TYPE ST_PNOutput_GenControl :
STRUCT
	w_Status					:	WORD;
	w_Warnings					:	WORD;
	w_Faults					:	WORD;
	ui_GeneratorStatus			:	UINT;	
END_STRUCT
END_TYPE

(* stored: Version 1.1.0.1, ProductVersion 3.1.4024.12
   DUT ST_PNOutput_GenControl: Id {8e5287c1-9f6f-4e04-8256-395225825020} *)
